(* CoDeSys 2.3.9.42 project: kod_zamok_89.pro *)
(* Libraries: Standard.lib 2.12.10 17:48:34, SYSLIBCALLBACK.LIB 2.12.10 17:48:32 *)

(* Global variable list: Global_Variables *)
VAR_GLOBAL
	s1, s2, s3, s4, s5, s6, s7, s8, s9: BOOL;
	start:BOOL;
	status:INT:=0;
END_VAR

(* POU PLC_PRG, ST *)
PROGRAM PLC_PRG
VAR
	enter: BOOL;
	mes: STRING;
END_VAR
(*первый этап*)
IF start=TRUE THEN
enter:=FALSE;
status:=0;
END_IF

(*второй этап*)
CASE status OF
0: IF s2 = TRUE THEN (*проверка-если кнопка №2 нажата, то status равен 1*)
status:=1;
ELSIF (s1 OR s3 OR s4 OR s5 OR s6 OR s7 OR s8 OR s9) = TRUE THEN (*если кнопки были нажаты ошибочно, то обнулять status*)
status:=0;
END_IF
1: IF s9 = TRUE THEN
status:=2;
ELSIF (s1 OR s3 OR s4 OR s5 OR s6 OR s7 OR s8) = TRUE THEN
status:=0;
END_IF
2: IF s1 = TRUE THEN
status:=3;
ELSIF (s1 OR s4 OR s5 OR s6 OR s7 OR s8) = TRUE THEN
status:=0;
END_IF
3: IF s6 = TRUE THEN
status:=4;
ELSIF (s4 OR s5 OR s7 OR s8) = TRUE THEN
status:=0;
END_IF
4: IF s7 = TRUE THEN
status:=5;
ELSIF (s4 OR s5 OR s8) = TRUE THEN
status:=0;
END_IF
END_CASE

(*заключение-вывод сообщение "замок открыт"*)
IF status=5 THEN
enter:=TRUE;
mes:='замок открыт';
ELSE
mes:='замок закрыт';
END_IF
END_PROGRAM

(* Visualisation visual
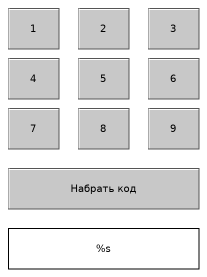
button at (50,40)-(101,81): text "1"; toggles .s1
button at (120,40)-(171,81): text "2"; toggles .s2
button at (190,40)-(241,81): text "3"; toggles .s3
button at (50,90)-(101,131): text "4"; toggles .s4
button at (120,90)-(171,131): text "5"; toggles .s5
button at (190,90)-(241,131): text "6"; toggles .s6
button at (50,140)-(101,181): text "7"; toggles .s7
button at (120,140)-(171,181): text "8"; toggles .s8
button at (190,140)-(241,181): text "9"; toggles .s9
button at (50,200)-(241,241): text "Набрать код"; taps .start
rectangle at (50,260)-(241,301): text "%s"; shows PLC_PRG.mes; alarm colour if PLC_PRG.enter
*)
